FUNCTION_BLOCK Dynamics
  (* Standard: 61499-2 *)
  (* Version 0.1, 2015-00-24, Jin, Jin-PC *)
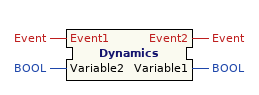
  EVENT_INPUT
    Event1;
  END_EVENT
  EVENT_OUTPUT
    Event2;
  END_EVENT
  VAR_INPUT
    Variable2 : BOOL;
  END_VAR
  VAR_OUTPUT
    Variable1 : BOOL;
  END_VAR
  EC_STATES
    Start;
  END_STATES
END_FUNCTION_BLOCK
